(*********************************** G.D S.p.A. - Technical Department ***********************************
============= PROGRAM INFO ============
FOLDER:             TBD
MACHINES INVOLVED:  TBD 

============= DESCRIPTION =============
csp machine declaration

============= REVISIONS ===============
Date		Version	 	Author      	Description             
----------	-------		------------  	--------------------------------------------
2019/04/05 	0000.00	 	M.Grasso		Creation of the PRG

**********************************************************************************************************)
(*$R process_ref := prc; $*)
PROGRAM csp_case_feed_shuttle_sensors_os
VAR
	
	prc:											process;
	prc_path:										STRING;
	
	part_present_di:								digital_input;
	
END_VAR

_read_var_input();

_object_manager();

IF NOT objects_running()
THEN
	RETURN;	
END_IF

_read_process_image();

_mode_manager();

_set_runtime_properties();

(********************************* BODY *********************************)
(************************************************************************)

_handle_messages();

_write_output();

ACTION _handle_messages:
;
END_ACTION

ACTION _handle_process_test:
;
END_ACTION

ACTION _mode_manager:
IF process_mode_req_is_pending(prc)
THEN
    process_apply_mode_req_first_step(prc);
    CASE process_get_mode(prc) OF
        MODE_TO_ABSENT:
			;
        MODE_TO_INACTIVE:
			;
        MODE_TO_TEST:
			;
        MODE_TO_OPERATIONAL:
			;
    END_CASE
    process_apply_mode_req_second_step(prc);
END_IF
END_ACTION

ACTION _object_manager:
IF objects_initialization()
THEN
	sub_process_init(
		object_name					:= 'csp_case_feed_shuttle_sensors_os.prc', 
		process						:= csp_case_feed_shuttle_sensors.prc, 
		CONVERSION_this				:= prc);
		
	prc_path 						:= process_get_path(prc);
	
	digital_input_init(
		object_name					:= CONCAT(prc_path, '_part_present_di'), 
		polarity_direct				:= TRUE, 
		process						:= prc, 
		CONVERSION_this				:= part_present_di);
	
END_IF

IF objects_running()
THEN
	process_cycle(prc);
END_IF
END_ACTION

ACTION _read_process_image:
;
END_ACTION

ACTION _read_var_input:
;
END_ACTION

ACTION _set_runtime_properties:
;
END_ACTION

ACTION _write_output:
;
END_ACTION

END_PROGRAM

(* stored: Version 1.1.0.1, ProductVersion 3.1.4024.3
   POU csp_case_feed_shuttle_sensors_os: Id {9d310f1d-9009-4c65-bf0d-7d85fe4873b4}, SpecialFunc None
   Action _handle_messages: Id {d1cf5af7-38da-4dee-a23b-70da2862556e}
   Action _handle_process_test: Id {92d177e7-d102-438a-afed-6e000dedd7a7}
   Action _mode_manager: Id {33cad1c0-393f-43ba-b328-9b2aa5f12be5}
   Action _object_manager: Id {54acb967-0c14-4b29-8764-3528a90ed67b}
   Action _read_process_image: Id {c869549b-8941-497c-b6e7-93a4f0aa8907}
   Action _read_var_input: Id {e8846e4c-8cce-4861-96b3-4c9f02e10ff6}
   Action _set_runtime_properties: Id {5f5cd86e-b71c-47c8-b965-e447358da85d}
   Action _write_output: Id {18e07d25-1303-4205-b4a3-c4804f595481} *)
